SUBAPPLICATION mapping_Uebung_016a (* Background Colour umschalten -- 3-fach *)
  (* Standard: 61499-2; Description: Copyright (c) 2023 Meisterschulen am Ostbahnhof This program and the accompanying materials are made available under the terms of the Eclipse Public License 2.0 which is available at https://www.eclipse.org/legal/epl-2.0/ SPDX-License-Identifier: EPL-2.0 *)
  (* Version 1.0, 2023-10-23, Franz Höpfinger, Meisterschulen am Ostbahnhof *)
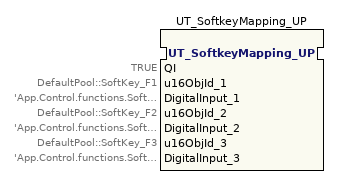
  FBS
    UT_SoftkeyMapping_UP : UT_SoftkeyMapping_UP(QI := TRUE, u16ObjId_1 := DefaultPool::SoftKey_F1, DigitalInput_1 := 'App.Control.functions.SoftKey_F1_UP', u16ObjId_2 := DefaultPool::SoftKey_F2, DigitalInput_2 := 'App.Control.functions.SoftKey_F2_UP', u16ObjId_3 := DefaultPool::SoftKey_F3, DigitalInput_3 := 'App.Control.functions.SoftKey_F3_UP');
  END_FBS
END_SUBAPPLICATION
